Staubli VAL3: start.pgx

program start()
begin
  //Here are examples for expansion addon functions.

  //
  title("Expansion examples")
  userPage()
  cls()
  //$getState
  call getState()
  //$delete
  call deleteFile()
  //$copy
  call copyFile()
  //$rename
  call renameFile()
  //$fileExists
  call fileExit()
  //$fileGet
  call fileRead()
  //$fileSet
  call fileWrite()
  //$getPowerCount
  call getPwrCnt()
  //$getFreeSpace
  call getMemoryFree()
  //$circleFind
  call fitCircle()
  //$setArmLimit,$setCellLimit
  call setLimit()
end
